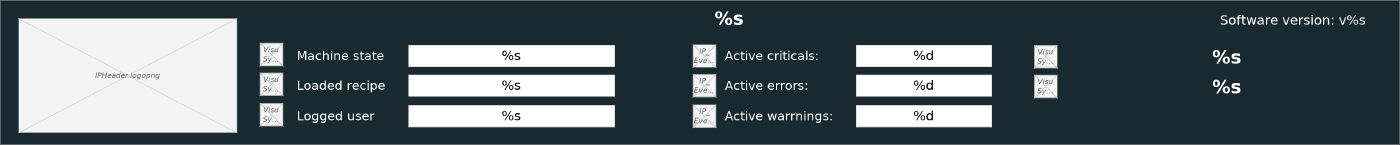
VISUALIZATION HeaderWinCE  // 1920x200
VAR_IN_OUT
	sMachineName		: STRING;					(*  *)
	sSoftwareVersion	: STRING;					(*  *)
	eMachineState		: E_MachineCtrlState;		(*  *)
	sCurrentRecipe		: STRING;					(*  *)
	sCurrentUser		: STRING;					(*  *)
	iActiveCriticals 	: UDINT;					(*  *)
	iActvieErrors		: UDINT;					(*  *)
	iActiveWarrnings	: UDINT;					(*  *)
	sCurrentDate		: STRING;					(*  *)
	sCurrentTime		: STRING;					(*  *)
END_VAR
    Label (404,59 133x36), "Machine state"
    Textfield (560,62 283x30), "%s", text list: 'TL_HeaderMachineState', text index: eMachineState
    Label (404,100 133x36), "Loaded recipe"
    Textfield (560,103 283x30), "%s", text variable: sCurrentRecipe
    Label (404,142 133x36), "Logged user"
    Textfield (560,145 283x30), "%s", text variable: sCurrentUser, text list: ''
    Label (991,59 133x36), "Active criticals:"
    Label (991,100 133x36), "Active errors:"
    Label (991,142 171x36), "Active warrnings:"
    Textfield (1174,62 186x30), "%d", text variable: iActiveCriticals
    Textfield (1174,103 186x30), "%d", text variable: iActvieErrors
    Textfield (1174,145 186x30), "%d", text variable: iActiveWarrnings
    Image (950,61 32x32), image: IP_EventSeverity.critical
    Image (950,102 32x32), image: IP_EventSeverity.error
    Image (950,144 32x32), image: IP_EventSeverity.warning
    Image (1418,62 32x32), image: VisuSymbols.Symbols.Calender
    Image (1418,103 32x32), image: VisuSymbols.Symbols.Clock
    Image (356,142 32x32), image: VisuSymbols.Symbols.User
    Image (356,59 32x32), image: VisuSymbols.Symbols.voltage
    Image (356,100 32x32), image: VisuSymbols.Symbols.Doc
    Textfield (700,10 600x30), "%s", text variable: sMachineName
    Textfield (1670,10 250x36), "Software version: v%s", text variable: sSoftwareVersion
    Textfield (1467,62 431x33), "%s", text variable: sCurrentDate
    Textfield (1467,103 431x33), "%s", text variable: sCurrentTime
    Image (25,25 300x158), image: IPHeader.logopng
END_VISUALIZATION

(* stored: Version 1.1.0.1, ProductVersion 3.1.4024.9
   Visu HeaderWinCE: Id {97ef52b6-4d62-4df4-91b8-3c212762baf0} *)
